RoboDK station: BaseOmronTM5-700.rdk

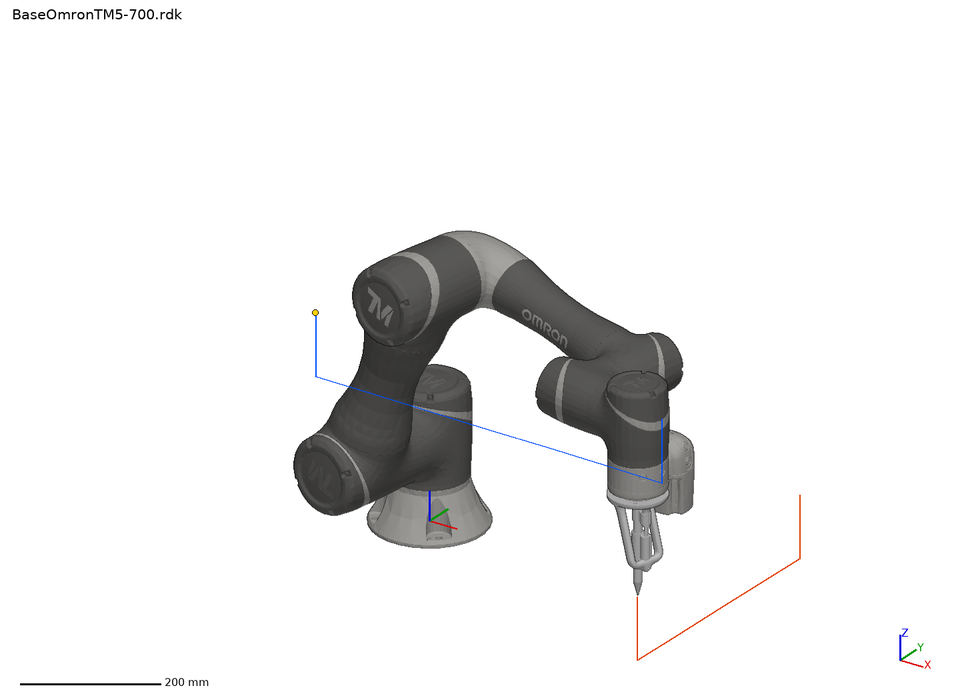
[picture v0: the station drawn from its stored meshes, robots at their saved joint values, targets as dots, program paths as lines]
Station BaseOmronTM5-700 (saved by RoboDK 5.6.7). Poses are relative to the parent item; angles as X-Y-Z fixed-axis rotations.
  - frame Omron TM5-700 Base at (0, 0, 0) mm
    - robot Omron TM5-700: 6 axes, payload 6 kg, reach 700 mm, repeatability 0.05 mm, weight 22.1 kg
        modified DH rows (alpha deg, a mm, theta deg, d mm): 0, 0, 0, 145.2; 90, 0, 90, 0; 0, 329, 0, 0; 0, 311, -90, 122.3; -90, 0, 0, 106.5; 90, 0, 180, 114.15
        joint limits [-270, -180, -155, -180, -180, -270] to [270, 180, 155, 180, 180, 270]; home [0, 0, 90, -90, 90, 0]; saved at [-8.675, 20.621, 83.138, -13.76, 90, -98.675]
      - tool PenHolderTCP, TCP at (0, 0, 165) mm, size 163 x 88.1 x 88.4 mm, geometry from PenHolderTCP.stl
    - frame Reference Rhino at (0, 0, 0) mm
      - object RhinoCrv at (0, 0, 0) mm
      - object testy at (0, 0, 0) mm, geometry from n     
  - machining project RhinoCrv Settings: rotZ(0) | rotX(0)*rotY(0) | rotz(0) | onStart | onPathStart | onApproach | onPoint | onRetract | onFinish | SetRPM(%1) | SetTool(%1) | Extruder(%1) | default | default | OutOnMov(%1) | OutOffMov(%1) | onPathFinish | M_RunCode(%1)
  - program BaseTest (19 instructions, listed below)
  - machining project testy Settings: rotZ(0) | rotX(0)*rotY(0) | rotz(0) | onStart | onPathStart | onApproach | onPoint | onRetract | onFinish | SetRPM(%1) | SetTool(%1) | Extruder(%1) | default | default | OutOnMov(%1) | OutOffMov(%1) | onPathFinish | M_RunCode(%1)
  - program testy (17 instructions, listed below)
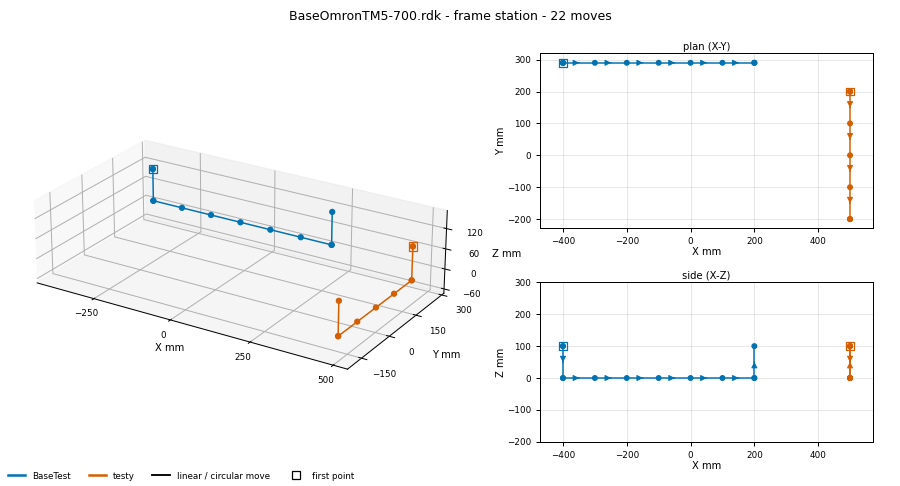
[picture p0: tool path of BaseOmronTM5-700.rdk in frame station, 22 of 22 moves have a stored position in this frame; points joined in program order, loops and branches not executed]

--- program BaseTest (robot Omron TM5-700) ---
  Smooth(1)
  Set speed (1000.0 mm/s)
  Set Ref.: Reference Rhino
  Set Tool: PenHolderTCP
  Show PenHolderTCP
  MoveJ 1 to (-400, 290, 100) mm, rotated rx 180 ry 0 rz 180 deg; joints [158.39, 12.914, 93.279, -16.193, 90, 68.39]
  MoveL 2 to (-400, 290, 100) mm, rotated rx 180 ry 0 rz 180 deg; joints [158.39, 12.914, 93.279, -16.193, 90, 68.39]
  MoveL 3 to (-400, 290, 0) mm, rotated rx 180 ry 0 rz 180 deg; joints [158.39, 20.403, 103.708, -34.111, 90, 68.39]
  MoveL 4 to (-400, 290, 0) mm, rotated rx 180 ry 0 rz 180 deg; joints [158.39, 20.403, 103.708, -34.111, 90, 68.39]
  Set speed (50.0 mm/s)
  MoveL 5 to (-300, 290, 0) mm, rotated rx 180 ry 0 rz 180 deg; joints [153.015, 8.295, 119.737, -38.032, 90, 63.015]
  MoveL 6 to (-200, 290, 0) mm, rotated rx 180 ry 0 rz 180 deg; joints [144.907, -3.275, 131.99, -38.715, 90, 54.907]
  MoveL 7 to (-100, 290, 0) mm, rotated rx 180 ry 0 rz 180 deg; joints [132.522, -12.99, 139.867, -36.877, 90, 42.522]
  MoveL 8 to (0, 290, 0) mm, rotated rx 180 ry 0 rz 180 deg; joints [114.943, -17.116, 142.589, -35.473, 90, 24.943]
  MoveL 9 to (100, 290, 0) mm, rotated rx 180 ry 0 rz 180 deg; joints [94.47, -12.99, 139.867, -36.877, 90, 4.47]
  MoveL 10 to (200, 290, 0) mm, rotated rx 180 ry 0 rz 180 deg; joints [75.722, -3.275, 131.99, -38.715, 90, -14.278]
  Set speed (1000.0 mm/s)
  MoveL 11 to (200, 290, 0) mm, rotated rx 180 ry 0 rz 180 deg; joints [75.722, -3.275, 131.99, -38.715, 90, -14.278]
  MoveL 12 to (200, 290, 100) mm, rotated rx 180 ry 0 rz 180 deg; joints [75.722, -13.157, 119.289, -16.132, 90, -14.278]

--- program testy (robot Omron TM5-700) ---
  Smooth(1)
  Set speed (1000.0 mm/s)
  Set Ref.: Reference Rhino
  Set Tool: PenHolderTCP
  Show PenHolderTCP
  MoveJ 1 to (500, 200, 100) mm, rotated rx -180 ry 0 rz -180 deg; joints [34.928, 20.621, 83.138, -13.76, 90, -55.072]
  MoveL 2 to (500, 200, 100) mm, rotated rx -180 ry 0 rz -180 deg; joints [34.928, 20.621, 83.138, -13.76, 90, -55.072]
  MoveL 3 to (500, 200, 0) mm, rotated rx -180 ry 0 rz -180 deg; joints [34.928, 27.212, 93.457, -30.669, 90, -55.072]
  MoveL 4 to (500, 200, 0) mm, rotated rx -180 ry 0 rz -180 deg; joints [34.928, 27.212, 93.457, -30.669, 90, -55.072]
  Set speed (50.0 mm/s)
  MoveL 5 to (500, 100, 0) mm, rotated rx -180 ry 0 rz -180 deg; joints [25.188, 22.826, 100.153, -32.979, 90, -64.812]
  MoveL 6 to (500, 0, 0) mm, rotated rx -180 ry 0 rz -180 deg; joints [14.158, 21.312, 102.387, -33.699, 90, -75.842]
  MoveL 7 to (500, -100, 0) mm, rotated rx -180 ry 0 rz -180 deg; joints [2.568, 22.826, 100.153, -32.979, 90, -87.432]
  MoveL 8 to (500, -200, 0) mm, rotated rx -180 ry 0 rz 180 deg; joints [-8.675, 27.212, 93.457, -30.669, 90, -98.675]
  Set speed (1000.0 mm/s)
  MoveL 9 to (500, -200, 0) mm, rotated rx -180 ry 0 rz 180 deg; joints [-8.675, 27.212, 93.457, -30.669, 90, -98.675]
  MoveL 10 to (500, -200, 100) mm, rotated rx -180 ry 0 rz 180 deg; joints [-8.675, 20.621, 83.138, -13.76, 90, -98.675]
